INTERFACE ITestEventHandler_UsesEventArgs EXTENDS IEventHandlerBase

METHOD OnThisEvent
VAR_INPUT
    EventArgs : IStreamReader;
END_VAR
END_METHOD

END_INTERFACE

(* stored: Version 1.1.0.1, ProductVersion 3.1.4024.4
   Itf ITestEventHandler_UsesEventArgs: Id {0053f9a9-a38e-487e-b30f-dd31d5ea3955}
   Method OnThisEvent: Id {f865e9f0-2f30-4b92-82cb-da64e51c58c9} *)
